{attribute addProperty BoxType "EP2816-0008-0016"}
{attribute addProperty Id "DO_Inputs_ChannelAT %I*ARRAY[0..1] OF DO_Inputs_Channel_AC4A9AF0128160DO_Inputs_DeviceAT %I*DO_Inputs_Device_213DCE554050DO_Outputs_ChannelAT %Q*ARRAY[0..1] OF DO_Outputs_Channel_33B76376128160DO_Outputs_DeviceAT %Q*DO_Outputs_Device_735003021620WcStateAT %I*WcState_F855686C1620InfoDataAT %I*InfoData_BC63D37F80100"}
{attribute addProperty CRC "1732962532"}
{attribute addProperty SizeInBites "408"}
{attribute addProperty SizeInBytes "51"}
TYPE EP2816_B01EBB0F :
STRUCT
	{attribute addProperty Name "DO_Inputs_Channel"}
	DO_Inputs_Channel : ARRAY[0..1] OF DO_Inputs_Channel_AC4A9AF0;
	{attribute addProperty Name "DO_Inputs_Device"}
	DO_Inputs_Device : DO_Inputs_Device_213DCE55;
	{attribute addProperty Name "DO_Outputs_Channel"}
	DO_Outputs_Channel : ARRAY[0..1] OF DO_Outputs_Channel_33B76376;
	{attribute addProperty Name "DO_Outputs_Device"}
	DO_Outputs_Device : DO_Outputs_Device_73500302;
	{attribute addProperty Name "WcState"}
	WcState : WcState_F855686C;
	{attribute addProperty Name "InfoData"}
	InfoData : InfoData_BC63D37F;
END_STRUCT
END_TYPE

(* stored: Version 1.2.0.0, ProductVersion 3.1.4024.9
   DUT EP2816_B01EBB0F: Id {95144b5f-a24a-42fc-a403-9da9d3c1bc8b} *)
